// TIA Portal V21 export
FUNCTION "Process_Data" : Void   // FC4, LAD
TITLE = PLC < - > CPC/CPLC data exchange
{ S7_Optimized_Access := 'TRUE' }
// Inputs:      Galileo -> PLC
// Outputs:  PLC -> Galileo
// stored: AutoNumber false, SetENOAutomatically false
   VAR_TEMP
      input : Byte;
   END_VAR
BEGIN

REGION Network 1: Input Byte 0 Rearm power C0 cabinet + Facility status
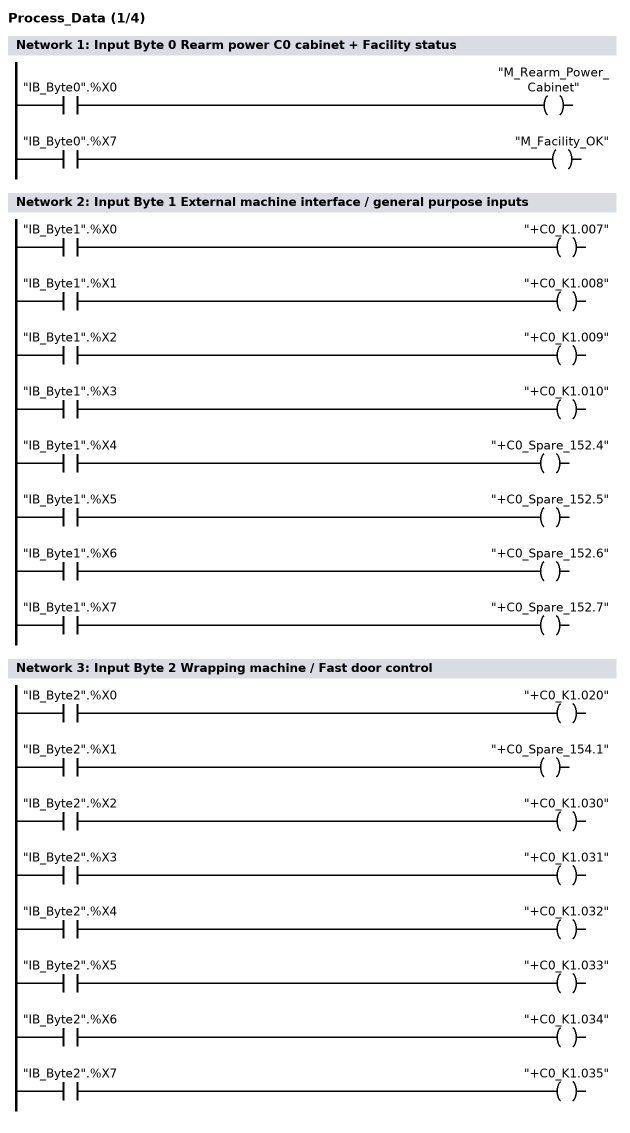
   RUNG wire#powerrail
      Contact( "IB_Byte0".%X0 )
      Coil( "M_Rearm_Power_Cabinet" )
   END_RUNG
   RUNG wire#powerrail
      Contact( "IB_Byte0".%X7 )
      Coil( "M_Facility_OK" )
   END_RUNG
   // the same network as SCL:
   "M_Rearm_Power_Cabinet" := "IB_Byte0".%X0;
   "M_Facility_OK" := "IB_Byte0".%X7;
END_REGION

REGION Network 2: Input Byte 1 External machine interface / general purpose inputs
   RUNG wire#powerrail
      Contact( "IB_Byte1".%X0 )
      Coil( "+C0_K1.007" )
   END_RUNG
   RUNG wire#powerrail
      Contact( "IB_Byte1".%X1 )
      Coil( "+C0_K1.008" )
   END_RUNG
   RUNG wire#powerrail
      Contact( "IB_Byte1".%X2 )
      Coil( "+C0_K1.009" )
   END_RUNG
   RUNG wire#powerrail
      Contact( "IB_Byte1".%X3 )
      Coil( "+C0_K1.010" )
   END_RUNG
   RUNG wire#powerrail
      Contact( "IB_Byte1".%X4 )
      Coil( "+C0_Spare_152.4" )
   END_RUNG
   RUNG wire#powerrail
      Contact( "IB_Byte1".%X5 )
      Coil( "+C0_Spare_152.5" )
   END_RUNG
   RUNG wire#powerrail
      Contact( "IB_Byte1".%X6 )
      Coil( "+C0_Spare_152.6" )
   END_RUNG
   RUNG wire#powerrail
      Contact( "IB_Byte1".%X7 )
      Coil( "+C0_Spare_152.7" )
   END_RUNG
   // the same network as SCL:
   "+C0_K1.007" := "IB_Byte1".%X0;
   "+C0_K1.008" := "IB_Byte1".%X1;
   "+C0_K1.009" := "IB_Byte1".%X2;
   "+C0_K1.010" := "IB_Byte1".%X3;
   "+C0_Spare_152.4" := "IB_Byte1".%X4;
   "+C0_Spare_152.5" := "IB_Byte1".%X5;
   "+C0_Spare_152.6" := "IB_Byte1".%X6;
   "+C0_Spare_152.7" := "IB_Byte1".%X7;
END_REGION

REGION Network 3: Input Byte 2 Wrapping machine / Fast door control
   RUNG wire#powerrail
      Contact( "IB_Byte2".%X0 )
      Coil( "+C0_K1.020" )
   END_RUNG
   RUNG wire#powerrail
      Contact( "IB_Byte2".%X1 )
      Coil( "+C0_Spare_154.1" )
   END_RUNG
   RUNG wire#powerrail
      Contact( "IB_Byte2".%X2 )
      Coil( "+C0_K1.030" )
   END_RUNG
   RUNG wire#powerrail
      Contact( "IB_Byte2".%X3 )
      Coil( "+C0_K1.031" )
   END_RUNG
   RUNG wire#powerrail
      Contact( "IB_Byte2".%X4 )
      Coil( "+C0_K1.032" )
   END_RUNG
   RUNG wire#powerrail
      Contact( "IB_Byte2".%X5 )
      Coil( "+C0_K1.033" )
   END_RUNG
   RUNG wire#powerrail
      Contact( "IB_Byte2".%X6 )
      Coil( "+C0_K1.034" )
   END_RUNG
   RUNG wire#powerrail
      Contact( "IB_Byte2".%X7 )
      Coil( "+C0_K1.035" )
   END_RUNG
   // the same network as SCL:
   "+C0_K1.020" := "IB_Byte2".%X0;
   "+C0_Spare_154.1" := "IB_Byte2".%X1;
   "+C0_K1.030" := "IB_Byte2".%X2;
   "+C0_K1.031" := "IB_Byte2".%X3;
   "+C0_K1.032" := "IB_Byte2".%X4;
   "+C0_K1.033" := "IB_Byte2".%X5;
   "+C0_K1.034" := "IB_Byte2".%X6;
   "+C0_K1.035" := "IB_Byte2".%X7;
END_REGION

REGION Network 4: Input Byte 3 Reset of safety zones
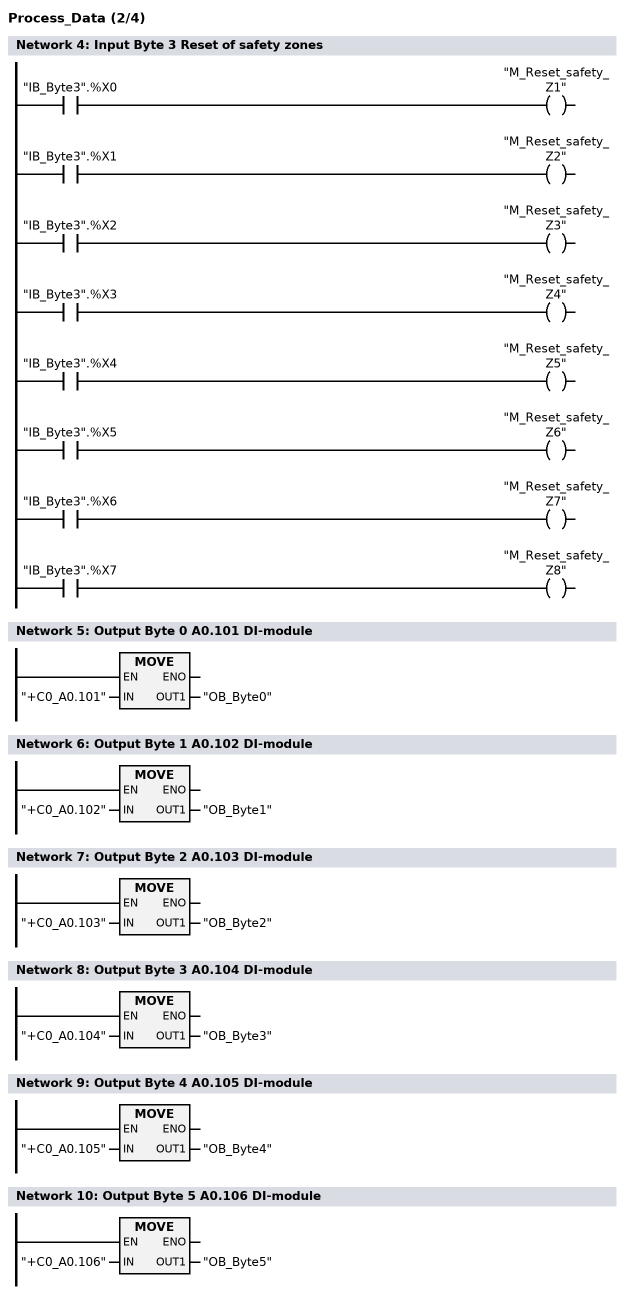
   RUNG wire#powerrail
      Contact( "IB_Byte3".%X0 )
      Coil( "M_Reset_safety_Z1" )
   END_RUNG
   RUNG wire#powerrail
      Contact( "IB_Byte3".%X1 )
      Coil( "M_Reset_safety_Z2" )
   END_RUNG
   RUNG wire#powerrail
      Contact( "IB_Byte3".%X2 )
      Coil( "M_Reset_safety_Z3" )
   END_RUNG
   RUNG wire#powerrail
      Contact( "IB_Byte3".%X3 )
      Coil( "M_Reset_safety_Z4" )
   END_RUNG
   RUNG wire#powerrail
      Contact( "IB_Byte3".%X4 )
      Coil( "M_Reset_safety_Z5" )
   END_RUNG
   RUNG wire#powerrail
      Contact( "IB_Byte3".%X5 )
      Coil( "M_Reset_safety_Z6" )
   END_RUNG
   RUNG wire#powerrail
      Contact( "IB_Byte3".%X6 )
      Coil( "M_Reset_safety_Z7" )
   END_RUNG
   RUNG wire#powerrail
      Contact( "IB_Byte3".%X7 )
      Coil( "M_Reset_safety_Z8" )
   END_RUNG
   // the same network as SCL:
   "M_Reset_safety_Z1" := "IB_Byte3".%X0;
   "M_Reset_safety_Z2" := "IB_Byte3".%X1;
   "M_Reset_safety_Z3" := "IB_Byte3".%X2;
   "M_Reset_safety_Z4" := "IB_Byte3".%X3;
   "M_Reset_safety_Z5" := "IB_Byte3".%X4;
   "M_Reset_safety_Z6" := "IB_Byte3".%X5;
   "M_Reset_safety_Z7" := "IB_Byte3".%X6;
   "M_Reset_safety_Z8" := "IB_Byte3".%X7;
END_REGION

REGION Network 5: Output Byte 0 A0.101 DI-module
   RUNG wire#powerrail
      Move(in := "+C0_A0.101", out1 => "OB_Byte0")
   END_RUNG
   // the same network as SCL:
   "OB_Byte0" := "+C0_A0.101";
END_REGION

REGION Network 6: Output Byte 1 A0.102 DI-module
   RUNG wire#powerrail
      Move(in := "+C0_A0.102", out1 => "OB_Byte1")
   END_RUNG
   // the same network as SCL:
   "OB_Byte1" := "+C0_A0.102";
END_REGION

REGION Network 7: Output Byte 2 A0.103 DI-module
   RUNG wire#powerrail
      Move(in := "+C0_A0.103", out1 => "OB_Byte2")
   END_RUNG
   // the same network as SCL:
   "OB_Byte2" := "+C0_A0.103";
END_REGION

REGION Network 8: Output Byte 3 A0.104 DI-module
   RUNG wire#powerrail
      Move(in := "+C0_A0.104", out1 => "OB_Byte3")
   END_RUNG
   // the same network as SCL:
   "OB_Byte3" := "+C0_A0.104";
END_REGION

REGION Network 9: Output Byte 4 A0.105 DI-module
   RUNG wire#powerrail
      Move(in := "+C0_A0.105", out1 => "OB_Byte4")
   END_RUNG
   // the same network as SCL:
   "OB_Byte4" := "+C0_A0.105";
END_REGION

REGION Network 10: Output Byte 5 A0.106 DI-module
   RUNG wire#powerrail
      Move(in := "+C0_A0.106", out1 => "OB_Byte5")
   END_RUNG
   // the same network as SCL:
   "OB_Byte5" := "+C0_A0.106";
END_REGION

REGION Network 11: Output Byte 6 A0.107 DI-module
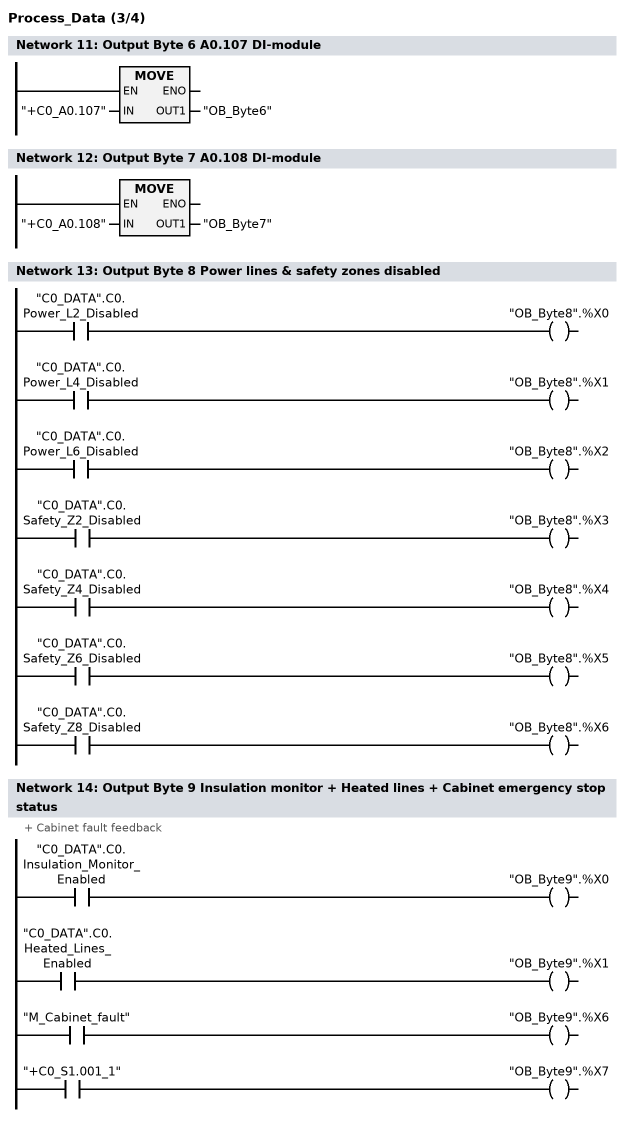
   RUNG wire#powerrail
      Move(in := "+C0_A0.107", out1 => "OB_Byte6")
   END_RUNG
   // the same network as SCL:
   "OB_Byte6" := "+C0_A0.107";
END_REGION

REGION Network 12: Output Byte 7 A0.108 DI-module
   RUNG wire#powerrail
      Move(in := "+C0_A0.108", out1 => "OB_Byte7")
   END_RUNG
   // the same network as SCL:
   "OB_Byte7" := "+C0_A0.108";
END_REGION

REGION Network 13: Output Byte 8 Power lines & safety zones disabled
   RUNG wire#powerrail
      Contact( "C0_DATA".C0.Power_L2_Disabled )
      Coil( "OB_Byte8".%X0 )
   END_RUNG
   RUNG wire#powerrail
      Contact( "C0_DATA".C0.Power_L4_Disabled )
      Coil( "OB_Byte8".%X1 )
   END_RUNG
   RUNG wire#powerrail
      Contact( "C0_DATA".C0.Power_L6_Disabled )
      Coil( "OB_Byte8".%X2 )
   END_RUNG
   RUNG wire#powerrail
      Contact( "C0_DATA".C0.Safety_Z2_Disabled )
      Coil( "OB_Byte8".%X3 )
   END_RUNG
   RUNG wire#powerrail
      Contact( "C0_DATA".C0.Safety_Z4_Disabled )
      Coil( "OB_Byte8".%X4 )
   END_RUNG
   RUNG wire#powerrail
      Contact( "C0_DATA".C0.Safety_Z6_Disabled )
      Coil( "OB_Byte8".%X5 )
   END_RUNG
   RUNG wire#powerrail
      Contact( "C0_DATA".C0.Safety_Z8_Disabled )
      Coil( "OB_Byte8".%X6 )
   END_RUNG
   // the same network as SCL:
   "OB_Byte8".%X0 := "C0_DATA".C0.Power_L2_Disabled;
   "OB_Byte8".%X1 := "C0_DATA".C0.Power_L4_Disabled;
   "OB_Byte8".%X2 := "C0_DATA".C0.Power_L6_Disabled;
   "OB_Byte8".%X3 := "C0_DATA".C0.Safety_Z2_Disabled;
   "OB_Byte8".%X4 := "C0_DATA".C0.Safety_Z4_Disabled;
   "OB_Byte8".%X5 := "C0_DATA".C0.Safety_Z6_Disabled;
   "OB_Byte8".%X6 := "C0_DATA".C0.Safety_Z8_Disabled;
END_REGION

REGION Network 14: Output Byte 9 Insulation monitor + Heated lines + Cabinet emergency stop status
   // + Cabinet fault feedback
   RUNG wire#powerrail
      Contact( "C0_DATA".C0.Insulation_Monitor_Enabled )
      Coil( "OB_Byte9".%X0 )
   END_RUNG
   RUNG wire#powerrail
      Contact( "C0_DATA".C0.Heated_Lines_Enabled )
      Coil( "OB_Byte9".%X1 )
   END_RUNG
   RUNG wire#powerrail
      Contact( "M_Cabinet_fault" )
      Coil( "OB_Byte9".%X6 )
   END_RUNG
   RUNG wire#powerrail
      Contact( "+C0_S1.001_1" )
      Coil( "OB_Byte9".%X7 )
   END_RUNG
   // the same network as SCL:
   "OB_Byte9".%X0 := "C0_DATA".C0.Insulation_Monitor_Enabled;
   "OB_Byte9".%X1 := "C0_DATA".C0.Heated_Lines_Enabled;
   "OB_Byte9".%X6 := "M_Cabinet_fault";
   "OB_Byte9".%X7 := "+C0_S1.001_1";
END_REGION

REGION Network 15: Output Byte 10 Emergency zones status
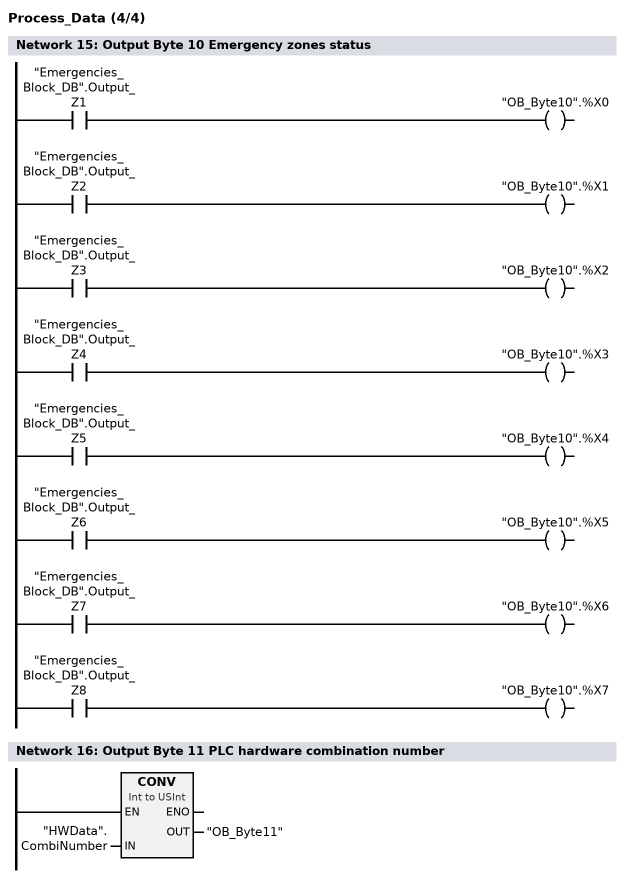
   RUNG wire#powerrail
      Contact( "Emergencies_Block_DB".Output_Z1 )
      Coil( "OB_Byte10".%X0 )
   END_RUNG
   RUNG wire#powerrail
      Contact( "Emergencies_Block_DB".Output_Z2 )
      Coil( "OB_Byte10".%X1 )
   END_RUNG
   RUNG wire#powerrail
      Contact( "Emergencies_Block_DB".Output_Z3 )
      Coil( "OB_Byte10".%X2 )
   END_RUNG
   RUNG wire#powerrail
      Contact( "Emergencies_Block_DB".Output_Z4 )
      Coil( "OB_Byte10".%X3 )
   END_RUNG
   RUNG wire#powerrail
      Contact( "Emergencies_Block_DB".Output_Z5 )
      Coil( "OB_Byte10".%X4 )
   END_RUNG
   RUNG wire#powerrail
      Contact( "Emergencies_Block_DB".Output_Z6 )
      Coil( "OB_Byte10".%X5 )
   END_RUNG
   RUNG wire#powerrail
      Contact( "Emergencies_Block_DB".Output_Z7 )
      Coil( "OB_Byte10".%X6 )
   END_RUNG
   RUNG wire#powerrail
      Contact( "Emergencies_Block_DB".Output_Z8 )
      Coil( "OB_Byte10".%X7 )
   END_RUNG
   // the same network as SCL:
   "OB_Byte10".%X0 := "Emergencies_Block_DB".Output_Z1;
   "OB_Byte10".%X1 := "Emergencies_Block_DB".Output_Z2;
   "OB_Byte10".%X2 := "Emergencies_Block_DB".Output_Z3;
   "OB_Byte10".%X3 := "Emergencies_Block_DB".Output_Z4;
   "OB_Byte10".%X4 := "Emergencies_Block_DB".Output_Z5;
   "OB_Byte10".%X5 := "Emergencies_Block_DB".Output_Z6;
   "OB_Byte10".%X6 := "Emergencies_Block_DB".Output_Z7;
   "OB_Byte10".%X7 := "Emergencies_Block_DB".Output_Z8;
END_REGION

REGION Network 16: Output Byte 11 PLC hardware combination number
   RUNG wire#powerrail
      { S7_Templates := "[SrcType := Int, DestType := USInt]" } Convert(in := "HWData".CombiNumber, out => "OB_Byte11")
   END_RUNG
   // the same network as SCL:
   "OB_Byte11" := INT_TO_USINT("HWData".CombiNumber);
END_REGION
END_FUNCTION
